FUNCTION_BLOCK FB68
TITLE = 'fault'
AUTHOR : CB

VAR
	fault_Z1 : FB50;
	fault_Z2 : FB57;
	fault_Z3 : FB63;
	fault_Z4 : FB67;
END_VAR


BEGIN


NETWORK
TITLE =
//
//	fault/fault_Z1
CALL #fault_Z1;



NETWORK
TITLE =
//
//	fault/fault_Z2
CALL #fault_Z2;



NETWORK
TITLE =
//
//	fault/fault_Z3
CALL #fault_Z3;



NETWORK
TITLE =
//
//	fault/fault_Z4
CALL #fault_Z4;




END_FUNCTION_BLOCK
